// TIA Portal V20 export
// export: Created 2025-12-01T14:57:43.8700533Z, ExportSetting None, DisplayName Totally Integrated Automation Portal, DisplayVersion V20 Update 3, DisplayName TIA Portal Openness, DisplayVersion V20 Update 3, DisplayName TIA Portal Version Control Interface, DisplayVersion V20 Update 3, DisplayName STEP 7 Professional, DisplayVersion V20 Update 3, DisplayName STEP 7 Safety, DisplayVersion V20 Update 2, DisplayName WinCC Basic/Comfort/Advanced, DisplayVersion V20 Update 3, DisplayName WinCC Professional, DisplayVersion V20 Update 3, DisplayName WinCC Unified, DisplayVersion V20 Update 3
FUNCTION "FC518_Funcion_Scanner" : Void   // FC518, LAD
{ S7_Optimized_Access := 'FALSE' }
AUTHOR : Nrodriguez
NAME : 20190926
VERSION : 1.1
// stored: AutoNumber false, SetENOAutomatically false
   VAR_INPUT
      NumeroMesa : UInt;
      Nodo_OK : Bool;
      Disparo_SCR : Bool;
      ID_Scanner : UInt;
      Byte_Ini_SCR : UInt;
      Porcentaje_XA_Error : UInt;
      Lecturas_seguidas_error : UInt;
   END_VAR
   VAR_TEMP
      Byte_Inicio : DWord;
      Aux_TOTAL : UDInt;
      Aux_Porcentaje : UInt;
      CERO : Byte;
      RETVALUE : Int;
   END_VAR
BEGIN

NETWORK
TITLE = Inicializacion
//==================================================================
// antes de hacer nada guardamos los valores de los ARs
// y la inicializacion de los datos

      L     0;
      T     #CERO;
      T     #Aux_Porcentaje;


//==================================================================

NETWORK
TITLE = Rearme del error de scanner y reinicio contadores de error
//=======================================================================
// si hay algún error relacionado con el scanner
// y pulsamos rearme, reseteamos el error y borramos
// los contadores de error

      SET;
      A(;
      O     "DB902_Estado_ZonaMesa".EstadoMesas[#NumeroMesa].Rearme_CBx;  // rearme de la mesa
      O     "DB902_Estado_ZonaMesa".EstadoMesas[#NumeroMesa].Resetear_CBx;
      O     "DB905_Estado_Escaners".Escaner[#ID_Scanner].orden_pantalla.reset;  // rearme de la pantalla
      );
      A     "DB905_Estado_Escaners".Escaner[#ID_Scanner].errores.Error_scanner;
      JC    rearmar_y_resetear;


//=======================================================================
// si no hemos saltado, seguimos con la ejecución normal del programa

      JU    comprobar_nodo;

//=======================================================================

rearmar_y_resetear:NOP   0;

// -- Reseteamos el error de la mesa
      SET;
      R     "DB900_Estado_Mesas".EstadoVI[#NumeroMesa].Err_SSCC_LectPorcentaje;
      R     "DB900_Estado_Mesas".EstadoVI[#NumeroMesa].Err_SSCC_LectConsecutiva;
      R     "DB900_Estado_Mesas".EstadoVI[#NumeroMesa].Err_Nodo_SSCC;
      R     "DB900_Estado_Mesas".EstadoVI[#NumeroMesa].Error_Mx;

// -- Reseteamos todos los errores del scanner en la pantalla
      CALL  FILL
      ( BVAL    := #CERO,
        RET_VAL := #RETVALUE,
        BLK     := "DB905_Estado_Escaners".Escaner[#ID_Scanner].errores
      );

// -- Reseteamos todos los contadores
// en vez de borrar todos los datos, inicializamos el valor de lecturas buenas a 100
// para que siga inmediatamente calculando porcentajes


      CALL  FILL
      ( BVAL    := #CERO,
        RET_VAL := #RETVALUE,
        BLK     := "DB216_Cnt_Estadisticas_Scanners".CNT_LectSCR[#ID_Scanner]
      );

// en vez de borrar todos los datos, inicializamos el valor de lecturas buenas a 100
// para que siga inmediatamente calculando porcentajes
      SET;
      L     100;
      T     "DB216_Cnt_Estadisticas_Scanners".CNT_LectSCR[#NumeroMesa].Lect_Good;

//=======================================================================
// -- guardamos los datos

      JU    Actualizar_datos;


//=======================================================================

NETWORK
TITLE = Comprobación de nodo presente para continuar con la ejecución.
//===================================================================================================================
// -- si no tenemos el nodo, solamente continuamos la ejecución
// -- si estamos con la simulación activa

comprobar_nodo:NOP   0;
      SET;
      AN    "Activar_Simulador";
      AN    #Nodo_OK;
      JC    generar_error;

      JU    disparar_Scanner;

generar_error:NOP   0;
      SET;
      S     "DB900_Estado_Mesas".EstadoVI[#NumeroMesa].Error_Mx;
      S     "DB900_Estado_Mesas".EstadoVI[#NumeroMesa].Err_Nodo_SSCC;
      S     "DB905_Estado_Escaners".Escaner[#ID_Scanner].errores.Error_reserva1;
      S     "DB905_Estado_Escaners".Escaner[#ID_Scanner].errores.Error_scanner;

      JU    Actualizar_datos;
//===================================================================================================================


NETWORK
TITLE = Disparo escaner
//===================================================================================================================
// calculamos la dirección donde está el scanner
disparar_Scanner:NOP   0;
      L     #Byte_Ini_SCR;  // calculo el puntero a la periferia
      L     1;
      +I;
      SLD   3;
      T     #Byte_Inicio;


//===================================================================================================================
      SET;
      O     "DB905_Estado_Escaners".Escaner[#ID_Scanner].orden_pantalla.disparo;  // si tengo disparo desde la pantalla
      O     #Disparo_SCR;  // si tenemos el disparo desde fuera
      JC    Disp;

// si no tenemos disparo tenemos que poner a cero el byte de disparo

      L     0;
      T     QB [#Byte_Inicio];
      JU    cont;


Disp: L     1;
      T     QB [#Byte_Inicio];
      JU    cont;

//===================================================================================================================

NETWORK
TITLE = comprobación de limites para generación de error
//===================================================================================================================
//Primero miramos si tenemos los datos suficientes como para generar el error de porcentaje. mínimo 60 lecturas
cont: NOP   0;

// NIEVES: LO PRIMERO QUE VAMOS A HACER ES COMPROBAR EL TOTAL DE LECTURAS.
// para evitar el peso de las lecturas antiguas en el calculo del porcentaje de error
// lo que vamos a hacer es movernos en un rango de lecturas de como máximo 500

// inicio revisión desbordamiento a 500

      L     "DB216_Cnt_Estadisticas_Scanners".CNT_LectSCR[#ID_Scanner].Lect_Good;
      L     "DB216_Cnt_Estadisticas_Scanners".CNT_LectSCR[#ID_Scanner].Lect_NoGood;
      +D;
      T     #Aux_TOTAL;

      SET;
      L     #Aux_TOTAL;
      L     500;
      <=I;
      JC    comprobacion;

// si hemos superado las 500 lecturas calculamos el porcentaje de error que llevamos

      L     "DB216_Cnt_Estadisticas_Scanners".CNT_LectSCR[#ID_Scanner].Lect_NoGood;
      ITD;
      L     DINT#100;
      *D;
      L     #Aux_TOTAL;
      /D;
      DTB;
      BTI;
      T     #Aux_Porcentaje;

// ahora que tenemos el porcentaje, dejamos la cantidad de lecturas buenas a 100 - porcentaje
// y las lecturas malas al mismo numero que el porcentaje

      L     #Aux_Porcentaje;
      T     "DB216_Cnt_Estadisticas_Scanners".CNT_LectSCR[#ID_Scanner].Lect_NoGood;

      L     100;
      L     #Aux_Porcentaje;
      -I;
      T     "DB216_Cnt_Estadisticas_Scanners".CNT_LectSCR[#ID_Scanner].Lect_Good;

      L     0;
      T     "DB216_Cnt_Estadisticas_Scanners".CNT_LectSCR[#ID_Scanner].Lect_NoFound;

// y volvemos a generar el total de lecturas con los parametros modificados

      L     "DB216_Cnt_Estadisticas_Scanners".CNT_LectSCR[#ID_Scanner].Lect_NoGood;
      L     "DB216_Cnt_Estadisticas_Scanners".CNT_LectSCR[#ID_Scanner].Lect_Good;
      +I;
      T     #Aux_TOTAL;

// fin revisión desbordamiento a 500


comprobacion:SET;
      L     #Aux_TOTAL;
      L     DINT#60;  // las 60 lecturas que consideramos como mínimo
      >=D;  // tenemos en cuenta que aprox 3 lecturas sean una tasa de error de 5% para ese minimo
      JC    calcular_porcentaje;

//==========================================================================================
// si no hemos saltado,  es porque no tenemos los datos suficientes para hacer ningun calculo
//pero pasamos a comprobar x cantidad de errores seguidos

      JU    Comprobar_errores_consecutivos;

//===================================================================================================================

NETWORK
TITLE = Comprobacion porcentaje de error

//==========================================================================================
// si tenemos los datos suficientes, pasamo a calcular el ratio de error

calcular_porcentaje:NOP   0;
      L     "DB216_Cnt_Estadisticas_Scanners".CNT_LectSCR[#ID_Scanner].Lect_NoGood;
      ITD;
      L     DINT#100;
      *D;
      L     #Aux_TOTAL;
      /D;
      DTB;
      BTI;
      T     #Aux_Porcentaje;

//==========================================================================================
// volcamos el dato del porcentaje en la pantalla para visualizarlo

      L     #Aux_Porcentaje;
      T     "DB216_Cnt_Estadisticas_Scanners".CNT_LectSCR[#ID_Scanner].Porcentaje_error_lecturas;


//==========================================================================================
// comparamos el porcentaje con el valor limite programado
      SET;
      L     #Porcentaje_XA_Error;
      L     #Aux_Porcentaje;
      >I;
      JC    porcentaje_correcto;
//==========================================================================================

// -- si no lo es, activamos el error correspondiente
      SET;
      S     "DB900_Estado_Mesas".EstadoVI[#NumeroMesa].Err_SSCC_LectConsecutiva;
      S     "DB900_Estado_Mesas".EstadoVI[#NumeroMesa].Error_Mx;
      S     "DB905_Estado_Escaners".Escaner[#ID_Scanner].errores.porcentaje;
      S     "DB905_Estado_Escaners".Escaner[#ID_Scanner].errores.Error_scanner;  // Error General Scanner

//==========================================================================================
porcentaje_correcto:NOP   0;
//==========================================================================================

NETWORK
TITLE = Comprobacion errores consecutivos
//==========================================================================================
// ahora vamos a controlar si aunque las estadisticas no sean malas,
// se están produciendo una serie de errores consecutivos

Comprobar_errores_consecutivos:NOP   0;

// al incrementar comprobamos si hemos llegado al máximo de seguidas configurado
      SET;
      L     "DB216_Cnt_Estadisticas_Scanners".CNT_LectSCR[#ID_Scanner].Lect_NoGood_consecutivas;
      L     #Lecturas_seguidas_error;
      <I;
      JC    Actualizar_datos;

// si no hemos saltado es que hay error.

      SET;
      S     "DB900_Estado_Mesas".EstadoVI[#NumeroMesa].Err_SSCC_LectConsecutiva;
      S     "DB900_Estado_Mesas".EstadoVI[#NumeroMesa].Error_Mx;
      S     "DB905_Estado_Escaners".Escaner[#ID_Scanner].errores.lecturas_consecuti;  // Error Porcentaje de lecturas correctas inferior al minimo
      S     "DB905_Estado_Escaners".Escaner[#ID_Scanner].errores.Error_scanner;  // Error General Scanner



NETWORK
TITLE = Actualización de los datos
//===================================================================================================================
// antes de salir de la función, actualizamos todos los datos
Actualizar_datos:NOP   0;

      CALL  BLKMOV
      ( SRCBLK  := "DB216_Cnt_Estadisticas_Scanners".CNT_LectSCR[#ID_Scanner],
        RET_VAL := #RETVALUE,
        DSTBLK  := "DB905_Estado_Escaners".Escaner[#ID_Scanner].contadores
      );


//+++++++++++++++++++++++++++++++++++++++++++++++++++++++++++++++++++++++++++
// sacar el dato del numero de la mesa

      L     #NumeroMesa;
      T     "DB905_Estado_Escaners".Escaner[#ID_Scanner].Numero_Mesa;





//===================================================================================================================
// -- recuperamos los valores de los ARs y salimos de la función.


END_FUNCTION
